Staubli VAL3: _endCycle.pjx

--- _endCycle.pjx ---
Parameters version=s7.7 stackSize=5000 millimeterUnit=true
Program file=start.pgx
Program file=stop.pgx
Data file=_endCycle.dtx
Library alias=cycleStatus path=Disk://cycleStatus/cycleStatus.pjx

--- start.pgx ---
public program start()
begin
  // end of cycle
  cycleStatus:bToEnd=true
  watch(cycleStatus:bToEnd==false,1)
end
